TYPE palletParamsL :
STRUCT
	

	zeroPos                  : REAL;
	size                     : REAL;

END_STRUCT
END_TYPE

(* stored: Version 1.1.0.1, ProductVersion 3.1.4024.3
   DUT palletParamsL: Id {50185d24-2309-4471-bbc3-c38785c4fbd6} *)
